# EPICS substitutions: opcpaepsApp/Db/eps_tmc.substitutions
file eps_tmc.template {
  pattern
    {PORT}
    {"EPS_ADS"}
}
